TYPE DUT_LoggerSample : STRUCT
    sample_index                 : UDINT;
    protocol_id                  : UINT;
    phase_id                     : UINT;
    angle_index                  : UINT;
    protocol2_local_sample_index : UINT;
    t_cycle_s                    : LREAL;
    experiment_angle_rad         : LREAL;
    x_ref_traj_m                 : LREAL;
    encoder_position_raw         : DINT;
    encoder_velocity_raw         : DINT;
    copley_actual_current_count  : INT;
    output_torque_count          : INT;
    fault_id                     : UDINT;
    iq_cmd_count_req_lreal       : LREAL;
    target_current_count_lreal   : LREAL;
END_STRUCT
END_TYPE

(* stored: Version 1.1.0.1, ProductVersion 3.1.4024.12
   DUT DUT_LoggerSample: Id {9f95b821-e6f9-4e51-98dd-900047a01007} *)
